{attribute 'GeneratedUsingTerminal: EK1122-0000-0018'}
{attribute addProperty BoxType "EK1122-0000-0018"}
{attribute addProperty Id "Beckhoff_EJ2xxxsub_EK1100EK1100_1FC0878B2"}
{attribute addProperty CRC "1399482409"}
{attribute addProperty Size "2"}
TYPE Beckhoff_EJ2xxxEK1122_536A6829 EXTENDS EK1122_1FC0878B :
STRUCT
	{attribute addProperty Name "Beckhoff_EJ2xxxsub_EK1100"}
	{attribute addProperty PreviousPort "Beckhoff EJ2xxxEK1122 : D"}
	Beckhoff_EJ2xxxsub_EK1100 : EK1100_1FC0878B;
END_STRUCT
END_TYPE

(* stored: Version 1.2.0.0, ProductVersion 3.1.4024.9
   DUT Beckhoff_EJ2xxxEK1122_536A6829: Id {2dd4fc41-8181-49f9-b95e-67308b3e5716} *)
